TYPE enum_E:
    (elit_Idle, elit_Off, elit_On, elit_Pushed, elit_Released, elit_Running, elit_s1, elit_s10, elit_s2, elit_s3, elit_s4, elit_s5, elit_s6, elit_s7, elit_s8, elit_s9);
END_TYPE

(* stored: ProductVersion 3.1.0.18, Version 1.1.0.1 *)
